PROGRAM Blinker
VAR
	fbMyBlinker	: FB_Blinker;
//	bBlink		: BOOL;
END_VAR


fbMyBlinker(tBlinkOn:= T#500MS, tBlinkOff:=T#3S);
bBlink	:= fbMyBlinker.Q;

IF bBlink = TRUE THEN
	rStatus	:= 1;
ELSE	
	rStatus	:= 0;
END_IF

END_PROGRAM

(* stored: Version 1.1.0.1
   POU Blinker: Id {7f134d98-dd2c-425e-a49e-7c64da5d2d98}, SpecialFunc None *)
